FUNCTION_BLOCK Double2Byte (* Basic Function Block Type *)
  (* Standard: 61499-2 *)
  (* Version 0.0, 12/6/2015, gulzha, nxtControl GmbH, Template *)
  PACKAGE Main;
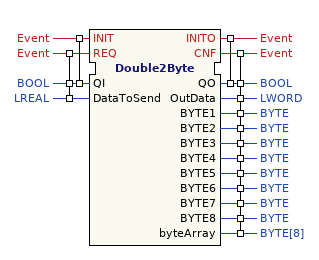
  EVENT_INPUT
    INIT WITH QI; (* Initialization Request *)
    REQ WITH QI, DataToSend; (* Normal Execution Request *)
  END_EVENT
  EVENT_OUTPUT
    INITO WITH QO; (* Initialization Confirm *)
    CNF WITH QO, OutData, BYTE1, BYTE2, BYTE3, BYTE4, BYTE5, BYTE6, BYTE7, BYTE8, byteArray; (* Execution Confirmation *)
  END_EVENT
  VAR_INPUT
    QI : BOOL; (* Input event qualifier *)
    DataToSend : LREAL;
  END_VAR
  VAR_OUTPUT
    QO : BOOL; (* Output event qualifier *)
    OutData : LWORD;
    BYTE1 : BYTE;
    BYTE2 : BYTE;
    BYTE3 : BYTE;
    BYTE4 : BYTE;
    BYTE5 : BYTE;
    BYTE6 : BYTE;
    BYTE7 : BYTE;
    BYTE8 : BYTE;
    byteArray : ARRAY [0..7] OF BYTE;
  END_VAR
  VAR
    temp : LWORD;
    i : INT;
    tempByte : BYTE;
  END_VAR
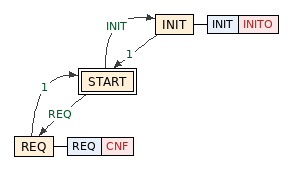
  EC_STATES
    START; (* Initial State *)
    INIT : INIT -> INITO; (* Initialization *)
    REQ : REQ -> CNF; (* Normal execution *)
  END_STATES
  EC_TRANSITIONS
    START TO INIT := INIT;
    INIT TO START := 1;
    START TO REQ := REQ;
    REQ TO START := 1;
  END_TRANSITIONS
  ALGORITHM INIT IN ST: (* Initialization algorithm *)
;
  END_ALGORITHM
  ALGORITHM REQ IN ST: (* Normally executed algorithm *)
;
temp := 0;
temp:= LREAL_TO_LWORD(DataToSend);


byteArray[0]:= LWORD_TO_BYTE(temp);
BYTE1 := byteArray[0];
temp:=  ROR(temp,8);

byteArray[1]:= LWORD_TO_BYTE(temp);
BYTE2 := byteArray[1];
temp:=  ROR(temp,8);

byteArray[2]:= LWORD_TO_BYTE(temp);
BYTE3 := byteArray[2];
temp:=  ROR(temp,8);

byteArray[3]:= LWORD_TO_BYTE(temp);
BYTE4 := byteArray[3];
temp:=  ROR(temp,8);

byteArray[4]:= LWORD_TO_BYTE(temp);
BYTE5 := byteArray[4];
temp:=  ROR(temp,8);

byteArray[5]:= LWORD_TO_BYTE(temp);
BYTE6 := byteArray[5];
temp:=  ROR(temp,8);

byteArray[6]:= LWORD_TO_BYTE(temp);
BYTE7 := byteArray[6];
temp:=  ROR(temp,8);

byteArray[7]:= LWORD_TO_BYTE(temp);
BYTE8 := byteArray[7];
temp:=  ROR(temp,8);

OutData:= temp; //DWORD_TO_LREAL(temp);
  END_ALGORITHM
END_FUNCTION_BLOCK
